(*
SPDX-FileCopyrightText: © 2026 Oleksandr Tiutyk <trofimich@gmail.com>
SPDX-License-Identifier: MIT
License: https://opensource.org/license/mit
*)

INTERFACE IDemoExceptionGenerator EXTENDS TOF_Automation.IInputLeafAutomationComponent

METHOD ThrowException
VAR_IN_OUT CONSTANT
	exceptionMessage : STRING(255);
	isCritical : BOOL; 
END_VAR
END_METHOD

END_INTERFACE

(* stored: Version 1.1.0.1
   Itf IDemoExceptionGenerator: Id {8e816f27-5e9e-40f4-870a-53e2b29bc372}
   Folder Commands: Id {e0a5b84a-d124-457e-8a7c-55aec22dd5c1}
   Method ThrowException: Id {e451ebad-6f63-4757-96ab-1019d494269c} *)
